FOR m := 0 TO 35 DO 
    b_A[m] := A[m];
END_FOR;
FOR m := 0 TO 5 DO 
    b_b_s[m] := 0.0;
    e[m] := 0.0;
    work[m] := 0.0;
END_FOR;
FOR m := 0 TO 35 DO 
    U[m] := 0.0;
    Vf[m] := 0.0;
END_FOR;
FOR m := 0 TO 4 DO 
    qq := (6 * m) + m;
    apply_transform := FALSE;
    nrm := xnrm2_l4(b_n := 6 - m, x := b_A, ix0 := qq + 1);
    IF nrm > 0.0 THEN 
        apply_transform := TRUE;
        IF b_A[qq] < 0.0 THEN 
            b_b_s[m] :=  -nrm;
        ELSE 
            b_b_s[m] := nrm;
        END_IF;
        IF ABS(b_b_s[m]) >= 1.0020841800044864E-292 THEN 
            i0_xscal_fiz1(b_n := 6 - m, a := 1.0 / b_b_s[m], x := b_A, ix0 := qq + 1);
        ELSE 
            qp1q := (qq - m) + 6;
            qjj := qq;
            WHILE (qjj + 1) <= qp1q DO
                b_A[qjj] := b_A[qjj] / b_b_s[m];
                qjj := qjj + 1;
            END_WHILE;
        END_IF;
        b_A[qq] := b_A[qq] + 1.0;
        b_b_s[m] :=  -b_b_s[m];
    ELSE 
        b_b_s[m] := 0.0;
    END_IF;
    qp1q := m + 1;
    WHILE (qp1q + 1) < 7 DO
        qjj := (6 * qp1q) + m;
        IF apply_transform THEN 
            temp16 := xdotc_iq(b_n := 6 - m, x := b_A, ix0 := qq + 1, y := b_A, iy0 := qjj + 1);
            i0_xaxpy_dmyz(b_n := 6 - m, a :=  -(temp16 / b_A[m + (6 * m)]), ix0 := qq + 1, y := b_A, iy0 := qjj + 1);
        END_IF;
        e[qp1q] := b_A[qjj];
        qp1q := qp1q + 1;
    END_WHILE;
    qq := m;
    WHILE (qq + 1) < 7 DO
        U[qq + (6 * m)] := b_A[(6 * m) + qq];
        qq := qq + 1;
    END_WHILE;
    IF (m + 1) <= 4 THEN 
        nrm := xnrm2_l4b(b_n := 5 - m, x := e, ix0 := m + 2);
        IF nrm = 0.0 THEN 
            e[m] := 0.0;
        ELSE 
            IF e[m + 1] < 0.0 THEN 
                e[m] :=  -nrm;
            ELSE 
                e[m] := nrm;
            END_IF;
            nrm := e[m];
            IF ABS(e[m]) >= 1.0020841800044864E-292 THEN 
                i0_xscal_fiz1t(b_n := 5 - m, a := 1.0 / e[m], x := e, ix0 := m + 2);
            ELSE 
                qq := m + 1;
                WHILE (qq + 1) <= 6 DO
                    e[qq] := e[qq] / nrm;
                    qq := qq + 1;
                END_WHILE;
            END_IF;
            e[m + 1] := e[m + 1] + 1.0;
            e[m] :=  -e[m];
            qq := m + 1;
            WHILE (qq + 1) < 7 DO
                work[qq] := 0.0;
                qq := qq + 1;
            END_WHILE;
            qq := m + 1;
            WHILE (qq + 1) < 7 DO
                i0_xaxpy_dmyzr(b_n := 5 - m, a := e[qq], x := b_A, ix0 := (m + (6 * qq)) + 2, y := work, iy0 := m + 2);
                qq := qq + 1;
            END_WHILE;
            qq := m + 1;
            WHILE (qq + 1) < 7 DO
                i0_xaxpy_dmyzr5(b_n := 5 - m, a := ( -e[qq]) / e[m + 1], x := work, ix0 := m + 2, y := b_A, iy0 := (m + (6 * qq)) + 2);
                qq := qq + 1;
            END_WHILE;
        END_IF;
        qq := m + 1;
        WHILE (qq + 1) < 7 DO
            Vf[qq + (6 * m)] := e[qq];
            qq := qq + 1;
        END_WHILE;
    END_IF;
END_FOR;
m := 4;
b_b_s[5] := b_A[35];
e[4] := b_A[34];
e[5] := 0.0;
FOR qq := 0 TO 5 DO 
    U[qq + 30] := 0.0;
END_FOR;
U[35] := 1.0;
FOR qp1q := 4 TO 0 BY -1 DO 
    qq := (6 * qp1q) + qp1q;
    IF b_b_s[qp1q] <> 0.0 THEN 
        qp1jj := qp1q + 1;
        WHILE (qp1jj + 1) < 7 DO
            qjj := ((6 * qp1jj) + qp1q) + 1;
            temp17 := xdotc_iq(b_n := 6 - qp1q, x := U, ix0 := qq + 1, y := U, iy0 := qjj);
            i0_xaxpy_dmyz(b_n := 6 - qp1q, a :=  -(temp17 / U[qq]), ix0 := qq + 1, y := U, iy0 := qjj);
            qp1jj := qp1jj + 1;
        END_WHILE;
        qjj := qp1q;
        WHILE (qjj + 1) < 7 DO
            qp1jj := (6 * qp1q) + qjj;
            U[qp1jj] :=  -U[qp1jj];
            qjj := qjj + 1;
        END_WHILE;
        U[qq] := U[qq] + 1.0;
        qq := 0;
        WHILE qq <= (qp1q - 1) DO
            U[qq + (6 * qp1q)] := 0.0;
            qq := qq + 1;
        END_WHILE;
    ELSE 
        FOR qjj := 0 TO 5 DO 
            U[qjj + (6 * qp1q)] := 0.0;
        END_FOR;
        U[qq] := 1.0;
    END_IF;
END_FOR;
FOR qq := 5 TO 0 BY -1 DO 
    IF (qq + 1) <= 4 THEN 
        IF e[qq] <> 0.0 THEN 
            qp1q := ((6 * qq) + qq) + 2;
            qjj := qq + 1;
            WHILE (qjj + 1) < 7 DO
                qp1jj := ((6 * qjj) + qq) + 2;
                temp18 := xdotc_iq(b_n := 5 - qq, x := Vf, ix0 := qp1q, y := Vf, iy0 := qp1jj);
                i0_xaxpy_dmyz(b_n := 5 - qq, a :=  -(temp18 / Vf[qp1q - 1]), ix0 := qp1q, y := Vf, iy0 := qp1jj);
                qjj := qjj + 1;
            END_WHILE;
        END_IF;
    END_IF;
    FOR qp1q := 0 TO 5 DO 
        Vf[qp1q + (6 * qq)] := 0.0;
    END_FOR;
    Vf[qq + (6 * qq)] := 1.0;
END_FOR;
FOR qq := 0 TO 5 DO 
    ztest := e[qq];
    IF b_b_s[qq] <> 0.0 THEN 
        rt := ABS(b_b_s[qq]);
        nrm := b_b_s[qq] / rt;
        b_b_s[qq] := rt;
        IF (qq + 1) < 6 THEN 
            ztest := ztest / nrm;
        END_IF;
        i0_xscal_fiz1t4(a := nrm, x := U, ix0 := (6 * qq) + 1);
    END_IF;
    IF (qq + 1) < 6 THEN 
        IF ztest <> 0.0 THEN 
            rt := ABS(ztest);
            nrm := rt / ztest;
            ztest := rt;
            b_b_s[qq + 1] := b_b_s[qq + 1] * nrm;
            i0_xscal_fiz1t4(a := nrm, x := Vf, ix0 := (6 * (qq + 1)) + 1);
        END_IF;
    END_IF;
    e[qq] := ztest;
END_FOR;
qq := 0;
nrm := 0.0;
FOR qp1q := 0 TO 5 DO 
    temp19 := ABS(b_b_s[qp1q]);
    temp20 := ABS(e[qp1q]);
    temp21 := MAX(temp19, temp20);
    nrm := MAX(nrm, temp21);
END_FOR;
WHILE ((m + 2) > 0) AND (qq < 75) DO
    qp1jj := m + 1;
    REPEAT 
        exitg1 := 0;
        qp1q := qp1jj;
        IF qp1jj = 0 THEN 
            exitg1 := 1;
        ELSE 
            rt := ABS(e[qp1jj - 1]);
            IF rt <= ((ABS(b_b_s[qp1jj - 1]) + ABS(b_b_s[qp1jj])) * 2.2204460492503131E-16) THEN 
                e[qp1jj - 1] := 0.0;
                exitg1 := 1;
            ELSIF (rt <= 1.0020841800044864E-292) OR ((qq > 20) AND (rt <= (2.2204460492503131E-16 * nrm))) THEN 
                e[qp1jj - 1] := 0.0;
                exitg1 := 1;
            ELSE 
                qp1jj := qp1jj - 1;
            END_IF;
        END_IF;
    UNTIL NOT(exitg1 = 0)
    END_REPEAT;
    IF (m + 1) = qp1jj THEN 
        qp1jj := 4;
    ELSE 
        qjj := m + 2;
        k_ii := m + 2;
        REPEAT 
            exitg1 := 0;
            IF k_ii >= qp1jj THEN 
                qjj := k_ii;
                IF k_ii = qp1jj THEN 
                    exitg1 := 1;
                ELSE 
                    rt := 0.0;
                    IF k_ii < (m + 2) THEN 
                        rt := ABS(e[k_ii - 1]);
                    END_IF;
                    IF k_ii > (qp1jj + 1) THEN 
                        rt := ABS(e[k_ii - 2]) + rt;
                    END_IF;
                    ztest := ABS(b_b_s[k_ii - 1]);
                    IF (ztest <= (2.2204460492503131E-16 * rt)) OR (ztest <= 1.0020841800044864E-292) THEN 
                        b_b_s[k_ii - 1] := 0.0;
                        exitg1 := 1;
                    ELSE 
                        k_ii := k_ii - 1;
                    END_IF;
                END_IF;
            ELSE 
                exitg1 := 1;
            END_IF;
        UNTIL NOT(exitg1 = 0)
        END_REPEAT;
        IF qjj = qp1jj THEN 
            qp1jj := 3;
        ELSIF (m + 2) = qjj THEN 
            qp1jj := 1;
        ELSE 
            qp1jj := 2;
            qp1q := qjj;
        END_IF;
    END_IF;
    CASE qp1jj OF
        1: 
            rt := e[m];
            e[m] := 0.0;
            qjj := m;
            WHILE (qjj + 1) >= (qp1q + 1) DO
                i0_xrotg(a := b_b_s[qjj], b := rt);
                ztest := i0_xrotg.c;
                sqds := i0_xrotg.b_s;
                IF (qjj + 1) > (qp1q + 1) THEN 
                    emm1 := e[qjj - 1];
                    rt := emm1 * ( -sqds);
                    e[qjj - 1] := emm1 * ztest;
                END_IF;
                i0_xrot_c5(x := Vf, ix0 := (6 * qjj) + 1, iy0 := (6 * (m + 1)) + 1, c := ztest, b_s := sqds);
                qjj := qjj - 1;
            END_WHILE;
        2: 
            rt := e[qp1q - 1];
            e[qp1q - 1] := 0.0;
            qjj := qp1q;
            WHILE (qjj + 1) <= (m + 2) DO
                i0_xrotg(a := b_b_s[qjj], b := rt);
                ztest := i0_xrotg.c;
                sqds := i0_xrotg.b_s;
                rt := ( -sqds) * e[qjj];
                e[qjj] := e[qjj] * ztest;
                i0_xrot_c5(x := U, ix0 := (6 * qjj) + 1, iy0 := (6 * (qp1q - 1)) + 1, c := ztest, b_s := sqds);
                qjj := qjj + 1;
            END_WHILE;
        3: 
            rt := b_b_s[m + 1];
            temp22 := ABS(rt);
            temp23 := ABS(b_b_s[m]);
            temp24 := MAX(temp22, temp23);
            temp25 := ABS(e[m]);
            temp26 := MAX(temp24, temp25);
            temp27 := ABS(b_b_s[qp1q]);
            temp28 := MAX(temp26, temp27);
            temp29 := ABS(e[qp1q]);
            ztest := MAX(temp28, temp29);
            rt := rt / ztest;
            smm1 := b_b_s[m] / ztest;
            emm1 := e[m] / ztest;
            sqds := b_b_s[qp1q] / ztest;
            smm1 := (((smm1 + rt) * (smm1 - rt)) + (emm1 * emm1)) / 2.0;
            emm1 := rt * emm1;
            emm1 := emm1 * emm1;
            IF (smm1 <> 0.0) OR (emm1 <> 0.0) THEN 
                shift := SQRT((smm1 * smm1) + emm1);
                IF smm1 < 0.0 THEN 
                    shift :=  -shift;
                END_IF;
                shift := emm1 / (smm1 + shift);
            ELSE 
                shift := 0.0;
            END_IF;
            rt := ((sqds + rt) * (sqds - rt)) + shift;
            ztest := (e[qp1q] / ztest) * sqds;
            qjj := qp1q + 1;
            WHILE qjj <= (m + 1) DO
                i0_xrotg(a := rt, b := ztest);
                sqds := i0_xrotg.c;
                smm1 := i0_xrotg.b_s;
                IF qjj > (qp1q + 1) THEN 
                    e[qjj - 2] := rt;
                END_IF;
                emm1 := e[qjj - 1];
                rt := b_b_s[qjj - 1];
                e[qjj - 1] := (emm1 * sqds) - (rt * smm1);
                ztest := smm1 * b_b_s[qjj];
                b_b_s[qjj] := b_b_s[qjj] * sqds;
                i0_xrot_c5(x := Vf, ix0 := (6 * (qjj - 1)) + 1, iy0 := (6 * qjj) + 1, c := sqds, b_s := smm1);
                b_b_s[qjj - 1] := (rt * sqds) + (emm1 * smm1);
                i0_xrotg(a := b_b_s[qjj - 1], b := ztest);
                sqds := i0_xrotg.c;
                smm1 := i0_xrotg.b_s;
                rt := (e[qjj - 1] * sqds) + (smm1 * b_b_s[qjj]);
                b_b_s[qjj] := (e[qjj - 1] * ( -smm1)) + (sqds * b_b_s[qjj]);
                ztest := smm1 * e[qjj];
                e[qjj] := e[qjj] * sqds;
                i0_xrot_c5(x := U, ix0 := (6 * (qjj - 1)) + 1, iy0 := (6 * qjj) + 1, c := sqds, b_s := smm1);
                qjj := qjj + 1;
            END_WHILE;
            e[m] := rt;
            qq := qq + 1;
        ELSE
            IF b_b_s[qp1q] < 0.0 THEN 
                b_b_s[qp1q] :=  -b_b_s[qp1q];
                i0_xscal_fiz1t4(a := -1.0, x := Vf, ix0 := (6 * qp1q) + 1);
            END_IF;
            qq := qp1q + 1;
            REPEAT 
                exitg1 := 0;
                IF (qp1q + 1) < 6 THEN 
                    IF b_b_s[qp1q] < b_b_s[qq] THEN 
                        rt := b_b_s[qp1q];
                        b_b_s[qp1q] := b_b_s[qq];
                        b_b_s[qq] := rt;
                        i0_xswap_gs(x := Vf, ix0 := (6 * qp1q) + 1, iy0 := (6 * (qp1q + 1)) + 1);
                        i0_xswap_gs(x := U, ix0 := (6 * qp1q) + 1, iy0 := (6 * (qp1q + 1)) + 1);
                        qp1q := qq;
                        qq := qq + 1;
                    ELSE 
                        exitg1 := 1;
                    END_IF;
                ELSE 
                    exitg1 := 1;
                END_IF;
            UNTIL NOT(exitg1 = 0)
            END_REPEAT;
            qq := 0;
            m := m - 1;
    END_CASE;
END_WHILE;
FOR m := 0 TO 5 DO 
    b_s[m] := b_b_s[m];
    FOR qq := 0 TO 5 DO 
        V[qq + (6 * m)] := Vf[(6 * m) + qq];
    END_FOR;
END_FOR;

END_FUNCTION_BLOCK

// ---- KinematicsForwAndInverseMatLab/xrot_c5.TcPOU
FUNCTION_BLOCK xrot_c5
VAR_INPUT
    ix0: DINT;
    iy0: DINT;
    c: LREAL;
    b_s: LREAL;
END_VAR
VAR_IN_OUT
    x: ARRAY [0..35] OF LREAL;
END_VAR
VAR_TEMP
    k: DINT;
    temp_tmp: DINT;
    temp_tmp_0: LREAL;
    temp_tmp_1: DINT;
    temp_tmp_2: LREAL;
END_VAR

FOR k := 0 TO 5 DO 
    temp_tmp := (iy0 + k) - 1;
    temp_tmp_0 := x[temp_tmp];
    temp_tmp_1 := (ix0 + k) - 1;
    temp_tmp_2 := x[temp_tmp_1];
    x[temp_tmp] := (temp_tmp_0 * c) - (temp_tmp_2 * b_s);
    x[temp_tmp_1] := (temp_tmp_2 * c) + (temp_tmp_0 * b_s);
END_FOR;

END_FUNCTION_BLOCK

// ---- KinematicsForwAndInverseMatLab/xswap_gs.TcPOU
FUNCTION_BLOCK xswap_gs
VAR_INPUT
    ix0: DINT;
    iy0: DINT;
END_VAR
VAR_IN_OUT
    x: ARRAY [0..35] OF LREAL;
END_VAR
VAR_TEMP
    temp: LREAL;
    k: DINT;
    temp_tmp: DINT;
    tmp: DINT;
END_VAR

FOR k := 0 TO 5 DO 
    temp_tmp := (ix0 + k) - 1;
    temp := x[temp_tmp];
    tmp := (iy0 + k) - 1;
    x[temp_tmp] := x[tmp];
    x[tmp] := temp;
END_FOR;

END_FUNCTION_BLOCK

// ---- KinematicsForwAndInverseMatLab/xscal_fiz1t4.TcPOU
FUNCTION_BLOCK xscal_fiz1t4
VAR_INPUT
    a: LREAL;
    ix0: DINT;
END_VAR
VAR_IN_OUT
    x: ARRAY [0..35] OF LREAL;
END_VAR
VAR_TEMP
    k: DINT;
END_VAR

k := ix0;
WHILE k <= (ix0 + 5) DO
    x[k - 1] := x[k - 1] * a;
    k := k + 1;
END_WHILE;

END_FUNCTION_BLOCK

// ---- KinematicsForwAndInverseMatLab/xaxpy_dmyz.TcPOU
FUNCTION_BLOCK xaxpy_dmyz
VAR_INPUT
    b_n: DINT;
    a: LREAL;
    ix0: DINT;
    iy0: DINT;
END_VAR
VAR_IN_OUT
    y: ARRAY [0..35] OF LREAL;
END_VAR
VAR_TEMP
    ix: DINT;
    iy: DINT;
    k: DINT;
END_VAR

IF (b_n >= 1) AND (a <> 0.0) THEN 
    ix := ix0 - 1;
    iy := iy0 - 1;
    k := 0;
    WHILE k <= (b_n - 1) DO
        y[iy] := (a * y[ix]) + y[iy];
        ix := ix + 1;
        iy := iy + 1;
        k := k + 1;
    END_WHILE;
END_IF;

END_FUNCTION_BLOCK

// ---- KinematicsForwAndInverseMatLab/xaxpy_dmyzr.TcPOU
FUNCTION_BLOCK xaxpy_dmyzr
VAR_INPUT
    b_n: DINT;
    a: LREAL;
    x: ARRAY [0..35] OF LREAL;
    ix0: DINT;
    iy0: DINT;
END_VAR
VAR_IN_OUT
    y: ARRAY [0..5] OF LREAL;
END_VAR
VAR_TEMP
    ix: DINT;
    iy: DINT;
    k: DINT;
END_VAR

IF (b_n >= 1) AND (a <> 0.0) THEN 
    ix := ix0 - 1;
    iy := iy0 - 1;
    k := 0;
    WHILE k <= (b_n - 1) DO
        y[iy] := (a * x[ix]) + y[iy];
        ix := ix + 1;
        iy := iy + 1;
        k := k + 1;
    END_WHILE;
END_IF;

END_FUNCTION_BLOCK

// ---- KinematicsForwAndInverseMatLab/xaxpy_dmyzr5.TcPOU
FUNCTION_BLOCK xaxpy_dmyzr5
VAR_INPUT
    b_n: DINT;
    a: LREAL;
    x: ARRAY [0..5] OF LREAL;
    ix0: DINT;
    iy0: DINT;
END_VAR
VAR_IN_OUT
    y: ARRAY [0..35] OF LREAL;
END_VAR
VAR_TEMP
    ix: DINT;
    iy: DINT;
    k: DINT;
END_VAR

IF (b_n >= 1) AND (a <> 0.0) THEN 
    ix := ix0 - 1;
    iy := iy0 - 1;
    k := 0;
    WHILE k <= (b_n - 1) DO
        y[iy] := (a * x[ix]) + y[iy];
        ix := ix + 1;
        iy := iy + 1;
        k := k + 1;
    END_WHILE;
END_IF;

END_FUNCTION_BLOCK

// ---- KinematicsForwAndInverseMatLab/xscal_fiz1t.TcPOU
FUNCTION_BLOCK xscal_fiz1t
VAR_INPUT
    b_n: DINT;
    a: LREAL;
    ix0: DINT;
END_VAR
VAR_IN_OUT
    x: ARRAY [0..5] OF LREAL;
END_VAR
VAR_TEMP
    b: DINT;
    k: DINT;
END_VAR

b := (ix0 + b_n) - 1;
k := ix0;
WHILE k <= b DO
    x[k - 1] := x[k - 1] * a;
    k := k + 1;
END_WHILE;

END_FUNCTION_BLOCK

// ---- KinematicsForwAndInverseMatLab/xscal_fiz1.TcPOU
FUNCTION_BLOCK xscal_fiz1
VAR_INPUT
    b_n: DINT;
    a: LREAL;
    ix0: DINT;
END_VAR
VAR_IN_OUT
    x: ARRAY [0..35] OF LREAL;
END_VAR
VAR_TEMP
    b: DINT;
    k: DINT;
END_VAR

b := (ix0 + b_n) - 1;
k := ix0;
WHILE k <= b DO
    x[k - 1] := x[k - 1] * a;
    k := k + 1;
END_WHILE;

END_FUNCTION_BLOCK

// ---- KinematicsForwAndInverseMatLab/xnrm2_l4.TcPOU
FUNCTION xnrm2_l4 : LREAL
VAR_INPUT
    b_n: DINT;
    x: ARRAY [0..35] OF LREAL;
    ix0: DINT;
END_VAR
VAR
    scale: LREAL;
    kend: DINT;
    absxk: LREAL;
    t: LREAL;
    k: DINT;
END_VAR

xnrm2_l4 := 0.0;
IF b_n >= 1 THEN 
    IF b_n = 1 THEN 
        xnrm2_l4 := ABS(x[ix0 - 1]);
    ELSE 
        scale := 3.3121686421112381E-170;
        kend := (ix0 + b_n) - 1;
        k := ix0;
        WHILE k <= kend DO
            absxk := ABS(x[k - 1]);
            IF absxk > scale THEN 
                t := scale / absxk;
                xnrm2_l4 := ((xnrm2_l4 * t) * t) + 1.0;
                scale := absxk;
            ELSE 
                t := absxk / scale;
                xnrm2_l4 := (t * t) + xnrm2_l4;
            END_IF;
            k := k + 1;
        END_WHILE;
        xnrm2_l4 := scale * SQRT(xnrm2_l4);
    END_IF;
END_IF;

END_FUNCTION

// ---- KinematicsForwAndInverseMatLab/xdotc_iq.TcPOU
FUNCTION xdotc_iq : LREAL
VAR_INPUT
    b_n: DINT;
    x: ARRAY [0..35] OF LREAL;
    ix0: DINT;
    y: ARRAY [0..35] OF LREAL;
    iy0: DINT;
END_VAR
VAR
    ix: DINT;
    iy: DINT;
    k: DINT;
END_VAR

xdotc_iq := 0.0;
IF b_n >= 1 THEN 
    ix := ix0;
    iy := iy0;
    k := 0;
    WHILE k <= (b_n - 1) DO
        xdotc_iq := (x[ix - 1] * y[iy - 1]) + xdotc_iq;
        ix := ix + 1;
        iy := iy + 1;
        k := k + 1;
    END_WHILE;
END_IF;

END_FUNCTION

// ---- KinematicsForwAndInverseMatLab/xnrm2_l4b.TcPOU
FUNCTION xnrm2_l4b : LREAL
VAR_INPUT
    b_n: DINT;
    x: ARRAY [0..5] OF LREAL;
    ix0: DINT;
END_VAR
VAR
    scale: LREAL;
    kend: DINT;
    absxk: LREAL;
    t: LREAL;
    k: DINT;
END_VAR

xnrm2_l4b := 0.0;
IF b_n >= 1 THEN 
    IF b_n = 1 THEN 
        xnrm2_l4b := ABS(x[ix0 - 1]);
    ELSE 
        scale := 3.3121686421112381E-170;
        kend := (ix0 + b_n) - 1;
        k := ix0;
        WHILE k <= kend DO
            absxk := ABS(x[k - 1]);
            IF absxk > scale THEN 
                t := scale / absxk;
                xnrm2_l4b := ((xnrm2_l4b * t) * t) + 1.0;
                scale := absxk;
            ELSE 
                t := absxk / scale;
                xnrm2_l4b := (t * t) + xnrm2_l4b;
            END_IF;
            k := k + 1;
        END_WHILE;
        xnrm2_l4b := scale * SQRT(xnrm2_l4b);
    END_IF;
END_IF;

END_FUNCTION

// ---- KinematicsForwAndInverseMatLab/isequal.TcPOU
FUNCTION isequal : BOOL
VAR_INPUT
    varargin_1: ARRAY [0..8] OF LREAL;
    varargin_2: ARRAY [0..8] OF LREAL;
END_VAR
VAR
    b_b_p: BOOL;
    k: DINT;
    exitg1: DINT;
END_VAR

isequal := FALSE;
b_b_p := TRUE;
k := 0;
REPEAT 
    exitg1 := 0;
    IF k < 9 THEN 
        IF varargin_1[k] <> varargin_2[k] THEN 
            b_b_p := FALSE;
            exitg1 := 1;
        ELSE 
            k := k + 1;
        END_IF;
    ELSE 
        exitg1 := 1;
    END_IF;
UNTIL NOT(exitg1 = 0)
END_REPEAT;
IF b_b_p THEN 
    isequal := TRUE;
END_IF;

END_FUNCTION

// ---- ServoControl/P_NormalizeJointVel.TcPOU
PROGRAM P_NormalizeJointVel
VAR
	fbActuatorVelToNormalized4 : FB_ActuatorVelFeedForward;
END_VAR


// Going from joint velocity to normalized signal inn PID
fbActuatorVelToNormalized4(fActuatorVelocity := G_InverseKinematics.fq4Dotref,
							fMaxActuatorVelocity := 0.030, //m/s
							fVelocityFeedForward => G_Servo.fNormalizedActuatorVelFeedForward_q4Dot);

END_PROGRAM

// ---- ServoControl/FB_ActuatorVelFeedForward.TcPOU
FUNCTION_BLOCK FB_ActuatorVelFeedForward
VAR_INPUT
	fActuatorVelocity : LREAL; //Input from inverse velocity kinematics
	fMaxActuatorVelocity : LREAL; //Actuator velocity at full joystick
END_VAR
VAR_OUTPUT
	fVelocityFeedForward : LREAL;
END_VAR
VAR
END_VAR


fVelocityFeedForward := fActuatorVelocity/fMaxActuatorVelocity;

END_FUNCTION_BLOCK

// ---- ServoControl/P_CarteseanControllerServoActuation4DOF.TcPOU
PROGRAM P_CarteseanControllerServoActuation4DOF
VAR
END_VAR



IF  G_Joystick.bJoystick2InUse OR G_Joystick.bJoystick3InUse OR G_Joystick.bJoystick4InUse OR G_Path.bPathActivated OR G_Heave.bHeaveActive  THEN
	
G_Servo.nServoPulseLenght1 := NormToPulseLenght(fJoyStickNormalized := G_Servo.f_u_q1,
								fEndPulseLengthPositive := 390, fStartPulseLengthPositive := 368, fStartPulseLengthNegative := 333, fEndPulseLengthNegative := 310);

G_Servo.nServoPulseLenght4 := NormToPulseLenght(fJoyStickNormalized := G_Servo.f_u_q2,
								fEndPulseLengthPositive := 410, fStartPulseLengthPositive := 360, fStartPulseLengthNegative := 340, fEndPulseLengthNegative := 290);

// Added minus on normalizsed signal for direction change on servo2, q3
G_Servo.nServoPulseLenght2 := NormToPulseLenght(fJoyStickNormalized := -G_Servo.f_u_q3,
								fEndPulseLengthPositive := 410, fStartPulseLengthPositive := 360, fStartPulseLengthNegative := 340, fEndPulseLengthNegative := 290);
//Telescope 					
G_Servo.nServoPulseLenght6 := NormToPulseLenght(fJoyStickNormalized := G_Servo.f_u_q4,
								fEndPulseLengthPositive := 450, fStartPulseLengthPositive := 360, fStartPulseLengthNegative := 330, fEndPulseLengthNegative := 250);
ELSE
G_Servo.nServoPulseLenght1 := 350;
G_Servo.nServoPulseLenght4 := 350;
G_Servo.nServoPulseLenght2 := 350;
G_Servo.nServoPulseLenght6 := 340;

END_IF



							
// Rotator
G_Servo.nServoPulseLenght3 := NormToPulseLenght(fJoyStickNormalized := G_Joystick.fJoystickRightNormalizedX,
								fEndPulseLengthPositive := 410, fStartPulseLengthPositive := 370, fStartPulseLengthNegative := 350, fEndPulseLengthNegative := 290);	
								
// Grasper
G_Servo.nServoPulseLenght5 := ButtonControlPulseLenght(fJoystickButtonFront := G_Buttons.bJoystickRightFrontEnable,
														fJoystickButtonBack := G_Buttons.bJoystickRightEnable,
															fNeutralPosition := 325);

END_PROGRAM

// ---- ServoControl/P_Idle.TcPOU
PROGRAM P_Idle
VAR
END_VAR

G_Servo.nServoPulseLenght1 := 350;
G_Servo.nServoPulseLenght2 := 350;
G_Servo.nServoPulseLenght3 := 350;
G_Servo.nServoPulseLenght4 := 350;
G_Servo.nServoPulseLenght5 := 335;
G_Servo.nServoPulseLenght6 := 340;

END_PROGRAM

// ---- HeaveCompensation/P_SetZero.TcPOU
PROGRAM P_SetZero
VAR
END_VAR

G_Heave.fThetaStart := G_SensorInput.fYRotDeg;
G_Toolpoint.fXref := G_Toolpoint.fX; //Set ref to actual
G_Toolpoint.fYref := G_Toolpoint.fY; //Set ref to actual
G_Toolpoint.fZref := G_Toolpoint.fZ; //Set ref to actual

END_PROGRAM

// ---- ControlBox/P_Outputs.TcPOU
PROGRAM P_Outputs
VAR
END_VAR

///////////////////// Lights //////////////////////////////


IF G_Buttons.bManualModeSelector OR G_Buttons.bAutoModeSelector THEN
	G_Outputs.bGreenButtonLight := FALSE;
	G_Outputs.bRedButtonLight := TRUE;
ELSE
	G_Outputs.bGreenButtonLight := TRUE;
	G_Outputs.bRedButtonLight := FALSE;
END_IF

END_PROGRAM

// ---- ControlBox/FB_AnalogInputScaling.TcPOU
FUNCTION_BLOCK FB_AnalogInputScaling
VAR_INPUT
	nRawInput 				: INT;
	stAnalogInputScaling    : ST_AnalogInputScaling;
END_VAR
VAR_OUTPUT
	fOutput 				: LREAL;
END_VAR
VAR
	fRawInput 				: LREAL;
	fNormalizedInput		: LREAL;
END_VAR

fRawInput := INT_TO_LREAL(nRawInput);

fNormalizedInput := (fRawInput - stAnalogInputScaling.fMinInputValue) / (stAnalogInputScaling.fMaxInputValue - stAnalogInputScaling.fMinInputValue);

fOutput := LIMIT(stAnalogInputScaling.fMinOutputValue, stAnalogInputScaling.fMinOutputValue + fNormalizedInput*(stAnalogInputScaling.fMaxOutputValue - stAnalogInputScaling.fMinOutputValue), stAnalogInputScaling.fMaxOutputValue);

END_FUNCTION_BLOCK

// ---- PathGenerator/P_PathGeneration.TcPOU
PROGRAM P_PathGeneration
VAR
	fbPathGenerator : FB_PathGenerator;
	Q1 : BOOL;
	ElapsedTime : LREAL;
	TimeX : LREAL := 2.5;
	TimeY : LREAL := 1.2;
	TimeZ : LREAL := 1.2;
	TimeEachSequence: INT;
	cartesianVelocity : LREAL;
END_VAR


cartesianVelocity := 0.050; // OPEN LOOP: Very much difference between 40 and 50

fbPathGenerator(bStart := G_Path.bStartPath, 
				TIN := T#40S , 
				Qout =>Q1, 
				t => ElapsedTime);


// -y, -halv z -halv y, + halv x + z, - halv y - halv x
IF ElapsedTime>= 0 AND ElapsedTime< 4 AND G_Path.bStartPath THEN 
	G_Path.bPathRunning := TRUE;
	G_Path.bPathFinnish := FALSE;
	G_InverseKinematics.fvXref := 0; //mm/S
	G_InverseKinematics.fvYref := -cartesianVelocity; //mm/S
	G_InverseKinematics.fvZref := 0; //mm/S
ELSIF ElapsedTime = 4 THEN
	G_Toolpoint.fXref := G_Toolpoint.fX; // RESET PATH TO CURRENT PATH IN TRANSITIONS
	G_Toolpoint.fYref := G_Toolpoint.fY;
	G_Toolpoint.fZref := G_Toolpoint.fZ;
ELSIF ElapsedTime> 4 AND ElapsedTime < 5 THEN
	G_InverseKinematics.fvXref := 0; //mm/S
	G_InverseKinematics.fvYref := 0; //mm/S
	G_InverseKinematics.fvZref := -cartesianVelocity; //mm/S
ELSIF ElapsedTime = 5 THEN
	G_Toolpoint.fXref := G_Toolpoint.fX; // RESET PATH TO CURRENT PATH IN TRANSITIONS
	G_Toolpoint.fYref := G_Toolpoint.fY;
	G_Toolpoint.fZref := G_Toolpoint.fZ;
ELSIF ElapsedTime> 5 AND ElapsedTime< 8 THEN
	G_InverseKinematics.fvXref := 0; //mm/S
	G_InverseKinematics.fvYref := cartesianVelocity; //mm/S
	G_InverseKinematics.fvZref := 0; //mm/S
ELSIF ElapsedTime = 8 THEN
	G_Toolpoint.fXref := G_Toolpoint.fX; // RESET PATH TO CURRENT PATH IN TRANSITIONS
	G_Toolpoint.fYref := G_Toolpoint.fY;
	G_Toolpoint.fZref := G_Toolpoint.fZ;
ELSIF ElapsedTime> 8 AND ElapsedTime< 10 THEN
	G_InverseKinematics.fvXref := cartesianVelocity; //mm/S
	G_InverseKinematics.fvYref := 0; //mm/S
	G_InverseKinematics.fvZref := 0; //mm/S
ELSIF ElapsedTime = 10 THEN
	G_Toolpoint.fXref := G_Toolpoint.fX; // RESET PATH TO CURRENT PATH IN TRANSITIONS
	G_Toolpoint.fYref := G_Toolpoint.fY;
	G_Toolpoint.fZref := G_Toolpoint.fZ;
ELSIF ElapsedTime = 10 THEN
	G_Toolpoint.fXref := G_Toolpoint.fX; // RESET PATH TO CURRENT PATH IN TRANSITIONS
	G_Toolpoint.fYref := G_Toolpoint.fY;
	G_Toolpoint.fZref := G_Toolpoint.fZ;
ELSIF ElapsedTime> 10 AND ElapsedTime< 12 THEN
	G_InverseKinematics.fvXref := 0; //mm/S
	G_InverseKinematics.fvYref := 0; //mm/S
	G_InverseKinematics.fvZref := cartesianVelocity; //mm/S
ELSIF ElapsedTime = 12 THEN
	G_Toolpoint.fXref := G_Toolpoint.fX; // RESET PATH TO CURRENT PATH IN TRANSITIONS
	G_Toolpoint.fYref := G_Toolpoint.fY;
	G_Toolpoint.fZref := G_Toolpoint.fZ;
ELSIF ElapsedTime> 12 AND ElapsedTime< 13 THEN
	G_InverseKinematics.fvXref := 0; //mm/S
	G_InverseKinematics.fvYref := -cartesianVelocity; //mm/S
	G_InverseKinematics.fvZref := 0; //mm/S
ELSIF ElapsedTime = 13 THEN
	G_Toolpoint.fXref := G_Toolpoint.fX; // RESET PATH TO CURRENT PATH IN TRANSITIONS
	G_Toolpoint.fYref := G_Toolpoint.fY;
	G_Toolpoint.fZref := G_Toolpoint.fZ;
ELSIF ElapsedTime> 13 AND ElapsedTime< 14 THEN
	G_InverseKinematics.fvXref := 0; //mm/S
	G_InverseKinematics.fvYref := 0; //mm/S
	G_InverseKinematics.fvZref := -cartesianVelocity; //mm/S
ELSIF ElapsedTime = 14 THEN
	G_Toolpoint.fXref := G_Toolpoint.fX; // RESET PATH TO CURRENT PATH IN TRANSITIONS
	G_Toolpoint.fYref := G_Toolpoint.fY;
	G_Toolpoint.fZref := G_Toolpoint.fZ;
ELSIF ElapsedTime> 14 AND ElapsedTime< 16 THEN
	G_InverseKinematics.fvXref := -cartesianVelocity; //mm/S
	G_InverseKinematics.fvYref := 0; //mm/S
	G_InverseKinematics.fvZref := 0; //mm/S

ELSE
	G_Path.bPathRunning := FALSE;
	G_Path.bPathFinnish := TRUE;
	G_Path.bStartPath := FALSE;
	ElapsedTime := 0;
	G_InverseKinematics.fvXref := 0; //mm/S
	G_InverseKinematics.fvYref := 0; //mm/S
	G_InverseKinematics.fvZref := 0; //mm/S
END_IF



(*
CASE CaseInt OF

1:  
fbPathGenerator(bStart := G_Path.bStartPath,
TIN := T#2S, 
Coordinate => G_InverseVelocityKinematics.fvXref, 
Qout => Q1);
IF Q1 THEN
	CaseInt:=2;
END_IF


2:     
fbPathGenerator2(bStart := G_Path.bStartPath,
TIN := T#2S, 
Coordinate => G_InverseVelocityKinematics.fvYref, 
Qout => Q2);
IF Q2 THEN
	CaseInt:=3;
END_IF

3:     
fbPathGenerator3(bStart := G_Path.bStartPath,
TIN := T#2S, 
Coordinate => G_InverseVelocityKinematics.fvZref, 
Qout => Q3);
IF Q3 THEN
	G_Path.bStartPath := FALSE;
	CaseInt:=1;
	Q1 := FALSE;
	Q2 := FALSE;
	Q3 := FALSE;
END_IF

END_CASE;

*)

END_PROGRAM

// ---- PathGenerator/P_PathGeneration_1.TcPOU
PROGRAM P_PathGeneration_1
VAR
	fbPathGenerator : FB_PathGenerator;
	Q1 : BOOL;
	ElapsedTime : LREAL;
	TimeX : LREAL := 2.5;
	TimeY : LREAL := 1.2;
	TimeZ : LREAL := 1.2;
	TimeEachSequence: INT;
	cartesianVelocity : LREAL;
END_VAR

// FOR  TELESCOPE TUNING

cartesianVelocity := 0.050; // OPEN LOOP: Very much difference between 40 and 50

fbPathGenerator(bStart := G_Path.bStartPath, 
				TIN := T#40S , 
				Qout =>Q1, 
				t => ElapsedTime);


IF ElapsedTime>= 0 AND ElapsedTime< 2 AND G_Path.bStartPath THEN 
	G_Path.bPathRunning := TRUE;
	G_Path.bPathFinnish := FALSE;
	G_InverseKinematics.fvXref := 0; //mm/S
	G_InverseKinematics.fvYref := -cartesianVelocity; //mm/S
	G_InverseKinematics.fvZref := 0; //mm/S
ELSIF ElapsedTime = 2 THEN
	G_Toolpoint.fXref := G_Toolpoint.fX; // RESET PATH TO CURRENT PATH IN TRANSITIONS
	G_Toolpoint.fYref := G_Toolpoint.fY;
	G_Toolpoint.fZref := G_Toolpoint.fZ;
ELSIF ElapsedTime> 2 AND ElapsedTime < 5 THEN
	G_InverseKinematics.fvXref := cartesianVelocity; //mm/S
	G_InverseKinematics.fvYref := 0; //mm/S
	G_InverseKinematics.fvZref := 0; //mm/S
ELSIF ElapsedTime = 5 THEN
	G_Toolpoint.fXref := G_Toolpoint.fX; // RESET PATH TO CURRENT PATH IN TRANSITIONS
	G_Toolpoint.fYref := G_Toolpoint.fY;
	G_Toolpoint.fZref := G_Toolpoint.fZ;
ELSIF ElapsedTime> 5 AND ElapsedTime < 8 THEN
	G_InverseKinematics.fvXref := 0; //mm/S
	G_InverseKinematics.fvYref := 0; //mm/S
	G_InverseKinematics.fvZref := cartesianVelocity; //mm/S
ELSIF ElapsedTime = 8 THEN
	G_Toolpoint.fXref := G_Toolpoint.fX; // RESET PATH TO CURRENT PATH IN TRANSITIONS
	G_Toolpoint.fYref := G_Toolpoint.fY;
	G_Toolpoint.fZref := G_Toolpoint.fZ;
ELSIF ElapsedTime> 8 AND ElapsedTime < 12 THEN
	G_InverseKinematics.fvXref := -cartesianVelocity; //mm/S
	G_InverseKinematics.fvYref := 0; //mm/S
	G_InverseKinematics.fvZref := 0; //mm/S
ELSIF ElapsedTime = 12 THEN
	G_Toolpoint.fXref := G_Toolpoint.fX; // RESET PATH TO CURRENT PATH IN TRANSITIONS
	G_Toolpoint.fYref := G_Toolpoint.fY;
	G_Toolpoint.fZref := G_Toolpoint.fZ;
ELSE
	G_Path.bPathRunning := FALSE;
	G_Path.bPathFinnish := TRUE;
	G_Path.bStartPath := FALSE;
	ElapsedTime := 0;
	G_InverseKinematics.fvXref := 0; //mm/S
	G_InverseKinematics.fvYref := 0; //mm/S
	G_InverseKinematics.fvZref := 0; //mm/S
END_IF



(*
CASE CaseInt OF

1:  
fbPathGenerator(bStart := G_Path.bStartPath,
TIN := T#2S, 
Coordinate => G_InverseVelocityKinematics.fvXref, 
Qout => Q1);
IF Q1 THEN
	CaseInt:=2;
END_IF


2:     
fbPathGenerator2(bStart := G_Path.bStartPath,
TIN := T#2S, 
Coordinate => G_InverseVelocityKinematics.fvYref, 
Qout => Q2);
IF Q2 THEN
	CaseInt:=3;
END_IF

3:     
fbPathGenerator3(bStart := G_Path.bStartPath,
TIN := T#2S, 
Coordinate => G_InverseVelocityKinematics.fvZref, 
Qout => Q3);
IF Q3 THEN
	G_Path.bStartPath := FALSE;
	CaseInt:=1;
	Q1 := FALSE;
	Q2 := FALSE;
	Q3 := FALSE;
END_IF

END_CASE;

*)

END_PROGRAM

// ---- PathGenerator/P_PathGeneration_3.TcPOU
PROGRAM P_PathGeneration_3
VAR
	fbPathGenerator : FB_PathGenerator;
	Q1 : BOOL;
	ElapsedTime : LREAL;
	TimeX : LREAL := 2.5;
	TimeY : LREAL := 1.2;
	TimeZ : LREAL := 1.2;
	TimeEachSequence: INT;
	cartesianVelocity : LREAL;
	timescaling: LREAL;
END_VAR

// FOR  TELESCOPE TUNING
timescaling := 3;
cartesianVelocity := 0.050/timescaling; // OPEN LOOP: Very much difference between 40 and 50 m/s

fbPathGenerator(bStart := G_Path.bStartPath, 
				TIN := T#150S , 
				Qout =>Q1, 
				t => ElapsedTime);


IF ElapsedTime>= 0*timescaling AND ElapsedTime< 2*timescaling AND G_Path.bStartPath THEN 
	G_Path.bPathRunning := TRUE;
	G_Path.bPathFinnish := FALSE;
	G_InverseKinematics.fvXref := cartesianVelocity; //mm/S
	G_InverseKinematics.fvYref := 0; //mm/S
	G_InverseKinematics.fvZref := 0; //mm/S
ELSIF ElapsedTime = 2*timescaling THEN
	G_Toolpoint.fXref := G_Toolpoint.fX; // RESET PATH TO CURRENT PATH IN TRANSITIONS
	G_Toolpoint.fYref := G_Toolpoint.fY;
	G_Toolpoint.fZref := G_Toolpoint.fZ;
ELSIF ElapsedTime> 2*timescaling AND ElapsedTime < 4*timescaling THEN
	G_InverseKinematics.fvXref := 0; //mm/S
	G_InverseKinematics.fvYref := cartesianVelocity; //mm/S
	G_InverseKinematics.fvZref := 0; //mm/S
ELSIF ElapsedTime = 4*timescaling THEN
	G_Toolpoint.fXref := G_Toolpoint.fX; // RESET PATH TO CURRENT PATH IN TRANSITIONS
	G_Toolpoint.fYref := G_Toolpoint.fY;
	G_Toolpoint.fZref := G_Toolpoint.fZ;
ELSIF ElapsedTime>= 4*timescaling AND ElapsedTime < 6*timescaling THEN
	G_InverseKinematics.fvXref := 0; //mm/S
	G_InverseKinematics.fvYref := 0; //mm/S
	G_InverseKinematics.fvZref := cartesianVelocity; //mm/S
ELSIF ElapsedTime = 6*timescaling THEN
	G_Toolpoint.fXref := G_Toolpoint.fX; // RESET PATH TO CURRENT PATH IN TRANSITIONS
	G_Toolpoint.fYref := G_Toolpoint.fY;
	G_Toolpoint.fZref := G_Toolpoint.fZ;
ELSIF ElapsedTime>= 6*timescaling AND ElapsedTime < 8*timescaling THEN
	G_InverseKinematics.fvXref := cartesianVelocity; //mm/S
	G_InverseKinematics.fvYref := -cartesianVelocity; //mm/S
	G_InverseKinematics.fvZref := 0; //mm/S
ELSIF ElapsedTime = 8*timescaling THEN
	G_Toolpoint.fXref := G_Toolpoint.fX; // RESET PATH TO CURRENT PATH IN TRANSITIONS
	G_Toolpoint.fYref := G_Toolpoint.fY;
	G_Toolpoint.fZref := G_Toolpoint.fZ;
ELSIF ElapsedTime>= 8*timescaling AND ElapsedTime < 13*timescaling THEN
	G_InverseKinematics.fvXref := 0; //mm/S
	G_InverseKinematics.fvYref := cartesianVelocity; //mm/S
	G_InverseKinematics.fvZref := 0; //mm/S
ELSIF ElapsedTime = 13*timescaling THEN
	G_Toolpoint.fXref := G_Toolpoint.fX; // RESET PATH TO CURRENT PATH IN TRANSITIONS
	G_Toolpoint.fYref := G_Toolpoint.fY;
	G_Toolpoint.fZref := G_Toolpoint.fZ;
ELSIF ElapsedTime>= 13*timescaling AND ElapsedTime < 17*timescaling THEN
	G_InverseKinematics.fvXref := -cartesianVelocity; //mm/S
	G_InverseKinematics.fvYref := -cartesianVelocity; //mm/S
	G_InverseKinematics.fvZref := 0; //mm/S
ELSIF ElapsedTime = 17*timescaling THEN
	G_Toolpoint.fXref := G_Toolpoint.fX; // RESET PATH TO CURRENT PATH IN TRANSITIONS
	G_Toolpoint.fYref := G_Toolpoint.fY;
	G_Toolpoint.fZref := G_Toolpoint.fZ;
ELSE
	G_Path.bPathRunning := FALSE;
	G_Path.bPathFinnish := TRUE;
	G_Path.bStartPath := FALSE;
	ElapsedTime := 0;
	G_InverseKinematics.fvXref := 0; //mm/S
	G_InverseKinematics.fvYref := 0; //mm/S
	G_InverseKinematics.fvZref := 0; //mm/S
END_IF



(*
CASE CaseInt OF

1:  
fbPathGenerator(bStart := G_Path.bStartPath,
TIN := T#2S, 
Coordinate => G_InverseVelocityKinematics.fvXref, 
Qout => Q1);
IF Q1 THEN
	CaseInt:=2;
END_IF


2:     
fbPathGenerator2(bStart := G_Path.bStartPath,
TIN := T#2S, 
Coordinate => G_InverseVelocityKinematics.fvYref, 
Qout => Q2);
IF Q2 THEN
	CaseInt:=3;
END_IF

3:     
fbPathGenerator3(bStart := G_Path.bStartPath,
TIN := T#2S, 
Coordinate => G_InverseVelocityKinematics.fvZref, 
Qout => Q3);
IF Q3 THEN
	G_Path.bStartPath := FALSE;
	CaseInt:=1;
	Q1 := FALSE;
	Q2 := FALSE;
	Q3 := FALSE;
END_IF

END_CASE;

*)

END_PROGRAM

// ---- POUs/P_SlaveInputControl.TcPOU
PROGRAM P_SlaveInputControl
VAR
	tempEncoder1 : LREAL := 0;
	tempEncoder11 : LREAL := 1;
END_VAR

END_PROGRAM

// ---- GlobalTextList.TcGTLO
TEXTLIST GlobalTextList
  568 = '%b'
  482 = '%f'
  171 = '%f '
  820 = 'Acknowledge'
  23 = 'Active'
  546 = 'AUTO'
  787 = 'CARTESIAN'
  890 = 'Drive STO'
  333 = 'EMG OK'
  810 = 'EMG Stop'
  911 = 'Finish'
  903 = 'Finnish'
  942 = 'Group'
  992 = 'Heave'
  176 = 'Heave Active'
  280 = 'IF RED LAMP: Sensors lost, '
  556 = 'IF RED LAMP: Sensors lost, reset slave arduino '
  705 = 'Inv Kinematics'
  419 = 'Inverse Kinematics'
  559 = 'joy sin'
  248 = 'JoyStick'
  839 = 'JoyStick or PATH'
  876 = 'MANUAL'
  88 = 'Manual Actuation Tests'
  792 = 'Manual Actuation Tests (enable in P_ModeControl)'
  998 = 'Manual Actuation Tests (first enable in P_ModeControl)'
  168 = 'Manual Actuation Tests (first enable P_ModeControl)'
  858 = 'MAX'
  712 = 'MIN'
  276 = 'Mode'
  730 = 'MODE'
  569 = 'NO KINEMATIC POS SOLUTION'
  704 = 'ON/OFF'
  365 = 'PATH      JOYSTICK'
  337 = 'Pos'
  773 = 'POS KIN SOLUTION'
  838 = 'Pos {f} [m]'
  623 = 'Pos {s} [m]'
  953 = 'PosRef'
  531 = 'PosRef {f} [m]'
  503 = 'PosRef {s} [m]'
  107 = 'PowerRefresh'
  729 = 'q1'
  291 = 'q1 [rad]'
  841 = 'q1PATH      JOYSTICK'
  753 = 'q2'
  755 = 'q2 [rad]'
  134 = 'q3'
  554 = 'q3 [rad]'
  914 = 'q4'
  435 = 'q4 [m]'
  949 = 'q4 [rad]'
  129 = 'Reset arduino'
  181 = 'Restart'
  267 = 'Run/Stop'
  955 = 'Running'
  791 = 'Sensors'
  131 = 'SENSORS LOST'
  147 = 'SINUS   JOYSTICK'
  603 = 'Solution found'
  649 = 'Start Path'
  940 = 'StartPath'
  92 = 'StartServo'
  501 = 'StartSinus'
  678 = 'TEMP FOR MAPPING pulse to encoder'
  384 = 'thetaDeg'
  488 = 'TwinSAFE'
  891 = 'VelRef'
  525 = 'VelRef [m/s]'
END_TEXTLIST

// ---- POUs/Visualization.TcVIS
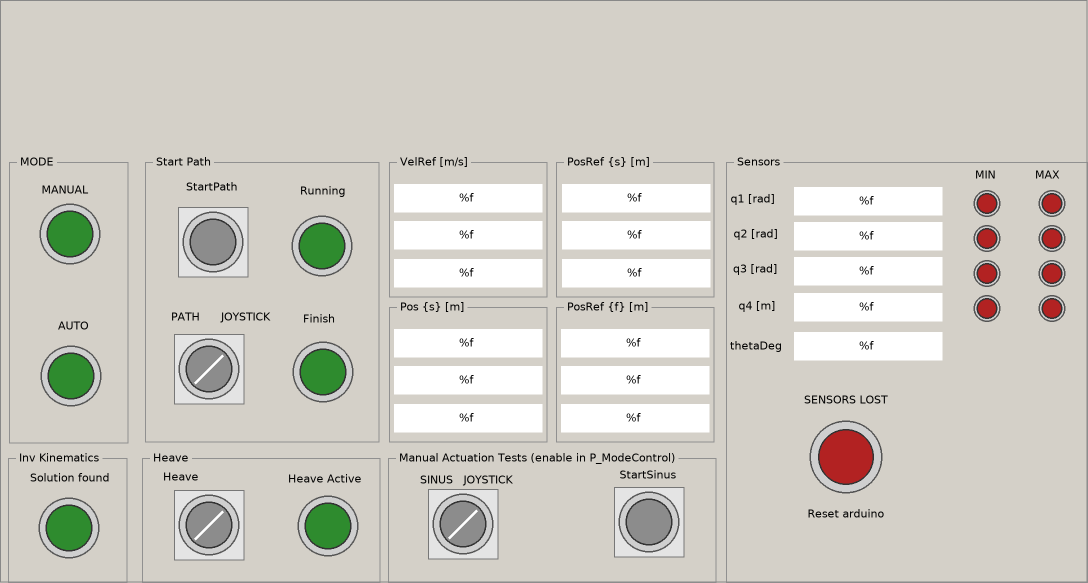
VISUALIZATION Visualization  // 1088x583
    GroupBox (388,450 328x133), "Manual Actuation Tests (enable in P_ModeControl)"
    GroupBox (389,154 158x143), "VelRef [m/s]"
        Label (99,258 150x30)
        Textfield (4,29 150x30), "%f", text variable: G_InverseKinematics.fvXref
        Textfield (4,66 150x30), "%f", text variable: G_InverseKinematics.fvYref
        Textfield (4,104 150x30), "%f", text variable: G_InverseKinematics.fvZref
    GroupBox (556,154 158x143), "PosRef {s} [m]"
        Textfield (5,29 150x30), "%f", text variable: G_Toolpoint.fXref
        Textfield (5,66 150x30), "%f", text variable: G_Toolpoint.fYref
        Textfield (5,104 150x30), "%f", text variable: G_Toolpoint.fZref
    GroupBox (389,299 158x143), "Pos {s} [m]"
        Textfield (4,29 150x30), "%f", text variable: G_Toolpoint.fX
        Textfield (4,66 150x30), "%f", text variable: G_Toolpoint.fY
        Textfield (4,104 150x30), "%f", text variable: G_Toolpoint.fZ
    GroupBox (9,154 119x289), "MODE"
        Lamp1 (26,45 70x70), variable: G_Buttons.bManualModeSelector, style: Lamp-Lamp1-Green
        Lamp1 (27,187 70x70), variable: G_Buttons.bAutoModeSelector, style: Lamp-Lamp1-Green
        Label (9,21 94x30), "MANUAL"
        Label (35,157 59x30), "AUTO"
    Label (113,154 150x30)
    GroupBox (145,154 234x288), "Start Path"
        Lamp1 (142,57 70x70), variable: G_Path.bPathRunning, style: Lamp-Lamp1-Green
        Lamp1 (143,183 70x70), variable: G_Path.bPathFinnish, style: Lamp-Lamp1-Green
        PushSwitch (33,53 70x70), variable: G_Path.bStartPath, behaviour: TOGGLE, style: Switch-PushSwitch-Gray
        Label (103,22 150x30), "Running"
        Label (99,150 150x30), "Finish"
        RotarySwitch (29,180 70x70), variable: G_Path.bPathActivated, behaviour: TOGGLE, style: Switch-RotarySwitch-Gray
        Label (7,148 137x30), "PATH JOYSTICK"
    Label (137,172 150x30), "StartPath"
    GroupBox (142,450 238x133), "Heave"
        Label (108,14 150x30), "Heave Active"
        RotarySwitch (32,40 70x70), variable: G_Heave.bHeaveEnable, behaviour: TOGGLE, style: Switch-RotarySwitch-Gray
        Lamp1 (151,41 70x70), variable: G_Heave.bHeaveActive, style: Lamp-Lamp1-Green
    Label (139,462 84x30), "Heave"
    GroupBox (8,450 119x133), "Inv Kinematics"
        Lamp1 (26,43 70x70), variable: G_InverseKinematics.bKinematicsSucsessful, style: Lamp-Lamp1-Green
        Label (16,13 92x30), "Solution found"
    GroupBox (726,154 362x429), "Sensors"
        Textfield (67,32 150x30), "%f", text variable: G_SensorsScaled.q1
        Textfield (67,67 150x30), "%f", text variable: G_SensorsScaled.q2
        Textfield (67,102 150x30), "%f", text variable: G_SensorsScaled.q3
        Textfield (67,138 150x30), "%f", text variable: G_SensorsScaled.q4
        Label (0,30 54x30), "q1 [rad]"
        Label (6,65 48x30), "q2 [rad]"
        Label (5,100 49x30), "q3 [rad]"
        Label (8,137 46x30), "q4 [m]"
        Label (104,181 150x30)
        Textfield (67,177 150x30), "%f", text variable: G_Heave.fTheta
        Label (0,177 60x30), "thetaDeg"
        Lamp1 (76,261 88x84), variable: G_SensorInput.bSensorDataLost, style: Lamp-Lamp1-Red
        Label (60,229 120x34), "SENSORS LOST"
        Label (60,343 120x34), "Reset arduino"
        Label (234,6 51x30), "MIN"
        Label (296,6 51x30), "MAX"
        Lamp1 (243,34 36x31), variable: G_ActuatorLimits.bq1Min, style: Lamp-Lamp1-Red
        Lamp1 (243,69 36x31), variable: G_ActuatorLimits.bq2Min, style: Lamp-Lamp1-Red
        Lamp1 (243,104 36x31), variable: G_ActuatorLimits.bq3Min, style: Lamp-Lamp1-Red
        Lamp1 (243,139 36x31), variable: G_ActuatorLimits.bq4Min, style: Lamp-Lamp1-Red
        Lamp1 (308,34 36x31), variable: G_ActuatorLimits.bq1Max, style: Lamp-Lamp1-Red
    Lamp1 (1034,223 36x31), variable: G_ActuatorLimits.bq2Max, style: Lamp-Lamp1-Red
    Lamp1 (1034,258 36x31), variable: G_ActuatorLimits.bq3Max, style: Lamp-Lamp1-Red
    Lamp1 (1034,293 36x31), variable: G_ActuatorLimits.bq4Max, style: Lamp-Lamp1-Red
    GroupBox (556,299 158x143), "PosRef {f} [m]"
        Textfield (4,29 150x30), "%f", text variable: G_Heave.r3x
        Textfield (4,66 150x30), "%f", text variable: G_Heave.r3y
        Textfield (4,104 150x30), "%f", text variable: G_Heave.r3z
    PushSwitch (614,487 70x70), variable: G_Servo.bStartSinus, behaviour: TOGGLE, style: Switch-PushSwitch-Gray
    Label (573,460 150x30), "StartSinus"
    RotarySwitch (428,489 70x70), variable: G_Servo.bSinusActive, behaviour: TOGGLE, style: Switch-RotarySwitch-Gray
    Label (398,465 137x30), "SINUS JOYSTICK"
END_VISUALIZATION
